TYPE
  (* Version 1.0, 2025-06-05, AK123700 *)
  message : STRUCT
    pubAdress : STRING;
    subAdress : STRING;
    msg : STRING;
  END_STRUCT;
END_TYPE
